FUNCTION InfluxAddData_1000Hz : BOOL
VAR_IN_OUT
	Data	: ST_DATA;
	DataCollector	: FB_InfluxDataCollector;
END_VAR

// =================== Test
	DataCollector.AddLreal(	'Test3',                                         Data.Gps.Inputs.x);

END_FUNCTION

(* stored: Version 1.1.0.1, ProductVersion 3.1.4022.11
   POU InfluxAddData_1000Hz: Id {42d4493b-eece-68f4-000d-07d00851ecfb}, SpecialFunc None *)
